INTERFACE I_Debug

END_INTERFACE

(* stored: Version 1.1.0.1
   Itf I_Debug: Id {72f669f1-a251-4fd7-81e9-899cb76da53c} *)
